// TwinCAT 3 PLC project PubSubSampleProject_Subscriber
// ProgramVersion: 3.1.4026.1+c9eadab3edd020c56c333d811d5b3c408c2550c8
// libraries:
//   Tc2_Standard, * (Beckhoff Automation GmbH)
//   Tc2_System, * (Beckhoff Automation GmbH)
// project tree:
//   DUTs/ ST_MyStructure.TcDUT
//   GVLs/ GVL_SubscriberVars_1.TcGVL, GVL_SubscriberVars_2.TcGVL (not stored)
//   / PlcTask.TcTTO
//   POUs/ MAIN.TcPOU
// (motion and I/O tree: see PLC project pubsubsampleproject_publisher)
// real-time tasks:
//   TASK PlcTask: cycle T#10ms, priority 20, ADS port 350
//   TASK PlcTask1: cycle T#10ms, priority 21, ADS port 351
// variable links:
//   PubSubSampleProject_Subscriber/PubSubSampleProject_Subscriber Instance <-> Device 1 (OPC UA RT)/Subscriber1/DsPubVars1
//     PlcTask Inputs/GVL_SubscriberVars_1.nCounter <-> Inputs/GVL_PublisherVars_1_nCounter
//     PlcTask Inputs/GVL_SubscriberVars_1.sString <-> Inputs/GVL_PublisherVars_1_sString
//     PlcTask Inputs/GVL_SubscriberVars_1.stMyStruct <-> Inputs/GVL_PublisherVars_1_stMyStruct
//   PubSubSampleProject_Subscriber/PubSubSampleProject_Subscriber Instance <-> Device 1 (OPC UA RT)/Subscriber2/DsPub1
//     PlcTask Inputs/GVL_SubscriberVars_2.nCounter <-> Inputs/GVL_PublisherVars_2_nCounter
//     PlcTask Inputs/GVL_SubscriberVars_2.sString <-> Inputs/GVL_PublisherVars_2_sString
//     PlcTask Inputs/GVL_SubscriberVars_2.stMyStruct <-> Inputs/GVL_PublisherVars_2_stMyStruct

CONFIGURATION PubSubSampleProject_Subscriber
    RESOURCE PLC ON TwinCAT3
        TASK PlcTask(INTERVAL := T#10ms, PRIORITY := 21);
        PROGRAM MAIN WITH PlcTask : MAIN;
    END_RESOURCE
END_CONFIGURATION

// ---- DUTs/ST_MyStructure.TcDUT
TYPE ST_MyStructure :
STRUCT
	a : INT;
	b : DINT;
	c : REAL;
	d : STRING(42);
END_STRUCT
END_TYPE

// ---- GVLs/GVL_SubscriberVars_1.TcGVL
{attribute 'qualified_only'}
(* This GVL contains variables that are defined as output variables for process image mapping *)
VAR_GLOBAL
	nCounter AT%I* : INT;
	sString AT%I* : STRING(42);
	stMyStruct AT%I* : ST_MyStructure;
END_VAR

// ---- POUs/MAIN.TcPOU
(* This sample demonstrates how to configure TF6105 OPC UA Pub/Sub with a publisher and a subscriber. This PLC Project contains the subscriber. *)
PROGRAM MAIN
VAR
END_VAR

END_PROGRAM
